INTERFACE I_Counter

METHOD IncCounter
VAR_INPUT
	Qty : INT;
END_VAR
END_METHOD

END_INTERFACE

(* stored: Version 1.1.0.1, ProductVersion 3.1.4024.12
   Itf I_Counter: Id {5abece88-5d7f-45fd-b04b-7ff1f352aa07}
   Method IncCounter: Id {587aeea1-538f-4e6d-9283-0ac292a00def} *)
